// Mitsubishi GX Works2 project: 逆物料方向顺序启动 - 顺物料方向顺序停止   PLC: FX1S

PROGRAM MAIN
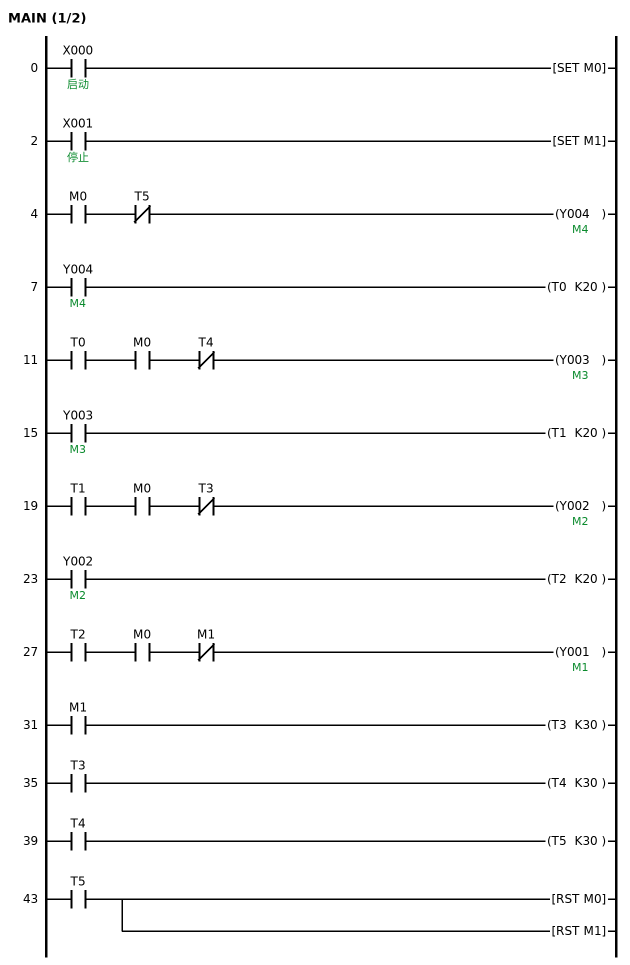
0     LD      X000  ; 启动
      SET     M0
2     LD      X001  ; 停止
      SET     M1
4     LD      M0
      ANI     T5
      OUT     Y004  ; M4
7     LD      Y004  ; M4
      OUT     T0 K20
11    LD      T0
      AND     M0
      ANI     T4
      OUT     Y003  ; M3
15    LD      Y003  ; M3
      OUT     T1 K20
19    LD      T1
      AND     M0
      ANI     T3
      OUT     Y002  ; M2
23    LD      Y002  ; M2
      OUT     T2 K20
27    LD      T2
      AND     M0
      ANI     M1
      OUT     Y001  ; M1
31    LD      M1
      OUT     T3 K30
35    LD      T3
      OUT     T4 K30
39    LD      T4
      OUT     T5 K30
43    LD      T5
      RST     M0
      RST     M1
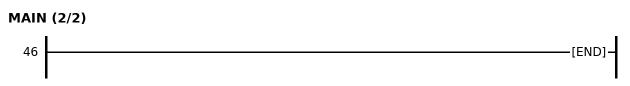
46    END
END_PROGRAM
